PROGRAM MAIN
VAR
	output1: BOOL;
	input1 : BOOL;
	andrew : DWORD;
	counter : Int;
END_VAR

counter := counter +1;

END_PROGRAM

(* stored: Version 1.1.0.1, ProductVersion 3.1.4024.12
   POU MAIN: Id {8d51e464-d0c5-46d7-9c54-d879937b15ac}, SpecialFunc None *)
